TYPE csp_case_loader_guide_accU_width_enum :
(
	CSP_CASE_LOADER_GUIDE_ACCU_WIDTH_STATUS_NOT_INITIALIZED 								:= 0,
	CSP_CASE_LOADER_GUIDE_ACCU_WIDTH_STATUS_DISABLED 										:= 10,
	CSP_CASE_LOADER_GUIDE_ACCU_WIDTH_STATUS_POSITION_CHECK									:= 20,
	CSP_CASE_LOADER_GUIDE_ACCU_WIDTH_STATUS_ENABLE_REQUEST 									:= 30,
	CSP_CASE_LOADER_GUIDE_ACCU_WIDTH_STATUS_ENABLED 										:= 40,
	CSP_CASE_LOADER_GUIDE_ACCU_WIDTH_STATUS_ABS_MOVE_REQUEST								:= 50,
	CSP_CASE_LOADER_GUIDE_ACCU_WIDTH_STATUS_ABS_MOVING										:= 60,
	CSP_CASE_LOADER_GUIDE_ACCU_WIDTH_STATUS_STOP_REQUEST 									:= 70,
	CSP_CASE_LOADER_GUIDE_ACCU_WIDTH_STATUS_DISABLE_REQUEST 								:= 80,
	CSP_CASE_LOADER_GUIDE_ACCU_WIDTH_STATUS_DISABLING 										:= 90
) := CSP_CASE_LOADER_GUIDE_ACCU_WIDTH_STATUS_NOT_INITIALIZED;
END_TYPE

(* stored: Version 1.1.0.1, ProductVersion 3.1.4022.18
   DUT csp_case_loader_guide_accU_width_enum: Id {fe3e7b76-cb10-4340-9031-85b1ba2439a9} *)
